FUNCTION_BLOCK FB_InstanceVariables

VAR
	test1, test2 : INT;
END_VAR

// This stays the same as the variable which we increment is reset on each call as its a var
test1 := M_AddLocal();

// This increases as the variable which we increment is added to the FB memory and is keep each cycle as its a var_inst
test2 := M_AddInst();

METHOD M_AddInst : INT

VAR_INST
	current : INT;
END_VAR
current := current + 1;

M_AddInst := current;
END_METHOD

METHOD M_AddLocal : INT

VAR
	current : INT;
END_VAR
current := current + 1;

M_AddLocal := current;
END_METHOD

END_FUNCTION_BLOCK

(* stored: Version 1.1.0.1
   POU FB_InstanceVariables: Id {674d412b-7505-49bb-99f4-82afc2d188be}, SpecialFunc None
   Method M_AddInst: Id {4e7dcfe1-1a73-439d-ac61-d87b8b66a59f}
   Method M_AddLocal: Id {1d602dc7-ea3b-4ef8-bdb4-da85fb83afb8} *)
